FUNCTION_BLOCK CameraMonitoring (* Tamplate for a simple Basic Function Block Type *)
  (* Standard: 61499-2 *)
  (* Version 0.0, 2018-03-05, 4DIAC-IDE, 4DIAC-Consortium *)
  (* Version 1.0, 2016-05-26, AZ, fortiss GmbH *)
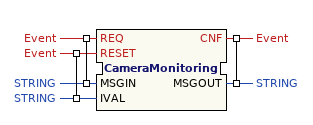
  EVENT_INPUT
    REQ WITH MSGIN; (* Normal Execution Request *)
    RESET WITH IVAL;
  END_EVENT
  EVENT_OUTPUT
    CNF WITH MSGOUT; (* Execution Confirmation *)
  END_EVENT
  VAR_INPUT
    MSGIN : STRING; (* Input event qualifier *)
    IVAL : STRING;
  END_VAR
  VAR_OUTPUT
    MSGOUT : STRING; (* Output event qualifier *)
  END_VAR
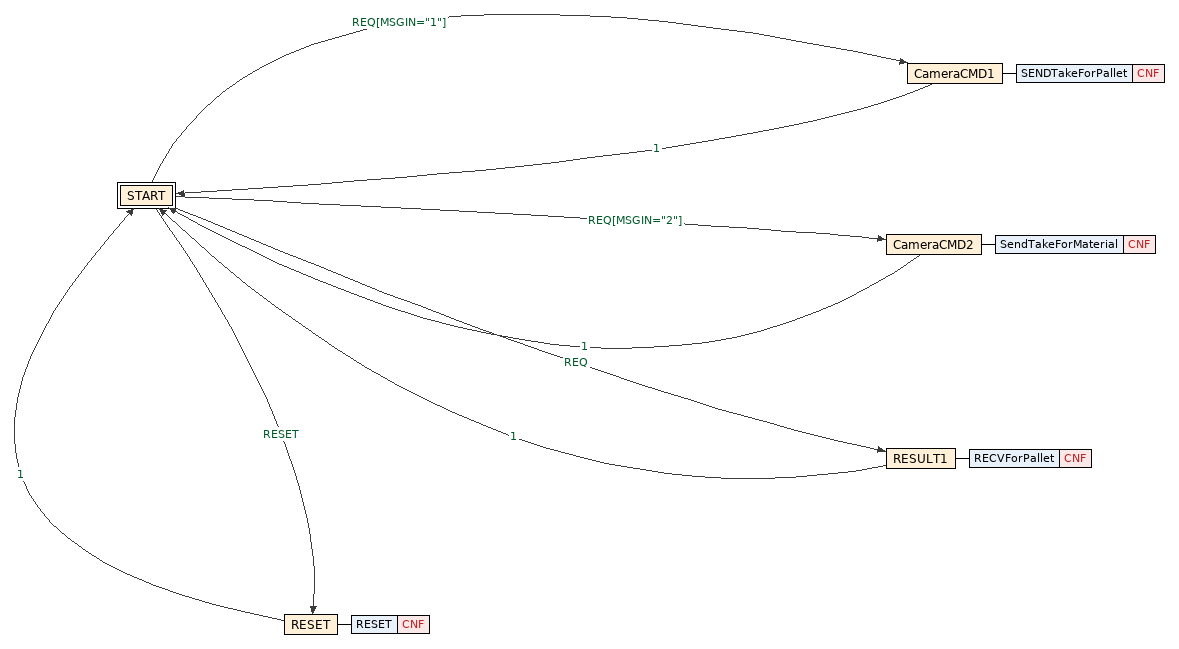
  EC_STATES
    START; (* Initial State *)
    CameraCMD1 : SENDTakeForPallet -> CNF;
    CameraCMD2 : SendTakeForMaterial -> CNF;
    RESULT1 : RECVForPallet -> CNF;
    RESET : RESET -> CNF;
  END_STATES
  EC_TRANSITIONS
    START TO CameraCMD1 := REQ[MSGIN="1"];
    CameraCMD1 TO START := 1;
    START TO CameraCMD2 := REQ[MSGIN="2"];
    CameraCMD2 TO START := 1;
    START TO RESULT1 := REQ;
    RESULT1 TO START := 1;
    START TO RESET := RESET;
    RESET TO START := 1;
  END_TRANSITIONS
  ALGORITHM SENDTakeForPallet IN ST: (* new algorithm *)
MSGOUT:="Taking photos for Pallet !";
  END_ALGORITHM
  ALGORITHM SendTakeForMaterial IN ST: (* new algorithm *)
MSGOUT:="Taking photos for Material !";
  END_ALGORITHM
  ALGORITHM RECVForPallet IN ST: (* new algorithm *)
MSGOUT:=MSGIN;
  END_ALGORITHM
  ALGORITHM RECVForMaterial IN ST: (* new algorithm *)
MSGOUT:=MSGIN;
  END_ALGORITHM
  ALGORITHM RESET IN ST: (* new algorithm *)
MSGOUT:=IVAL;
  END_ALGORITHM
END_FUNCTION_BLOCK
